(* IEC 61131-3 sources: RL_MAR/experiments/comparison/llm4plc/results/gpt-4o-mini_20260506_100619/20260506_101515, 1 file *)

(* ---- generated_code_iteration_0.st ---- *)
ructured-text
START_ST
FUNCTION_BLOCK WastewaterControl
VAR_INPUT
    InFlow : REAL;
    OutFlow : REAL;
    pH : REAL;
    TankLvl : REAL;
END_VAR

VAR_OUTPUT
    Pump1 : BOOL;
    Pump2 : BOOL;
    Valve1 : BOOL;
    Valve2 : BOOL;
END_VAR

VAR
    LowInFlow : REAL := 100.0;
    HighOutFlow : REAL := 90.0;
    DesiredPH : REAL := 7.0;
    HighTankLvl : REAL := 80.0;
    state : INT; // THE STATE VARIABLE
    prevState : INT; // THE PREVIOUS STATE VARIABLE
END_VAR

// STATE 0: INITIALIZE
IF state = 0 THEN
    Pump1 := FALSE;
    Pump2 := FALSE;
    Valve1 := FALSE;
    Valve2 := FALSE;
    state := 1; // Transition to CONTROL_PUMPS
END_IF

// STATE 1: CONTROL_PUMPS
IF state = 1 THEN
    IF InFlow < LowInFlow THEN
        Pump1 := TRUE; // Turn on Pump1
    ELSE
        Pump1 := FALSE; // Turn off Pump1
    END_IF;

    IF OutFlow > HighOutFlow THEN
        Pump2 := TRUE; // Turn on Pump2
    ELSE
        Pump2 := FALSE; // Turn off Pump2
    END_IF;

    state := 2; // Transition to CONTROL_VALVES
END_IF

// STATE 2: CONTROL_VALVES
IF state = 2 THEN
    IF pH < DesiredPH THEN
        Valve1 := TRUE; // Open Valve1
    ELSE
        Valve1 := FALSE; // Close Valve1
    END_IF;

    IF TankLvl > HighTankLvl THEN
        Valve2 := TRUE; // Open Valve2
    ELSE
        Valve2 := FALSE; // Close Valve2
    END_IF;

    // Optionally, return to state 1 or remain in state 2 based on conditions
    state := 1; // For continuous control, loop back to CONTROL_PUMPS
END_IF

END_FUNCTION_BLOCK
END_ST
